(* IEC 61131-3 sources: eCockpitGit/test_project/src/%F%00 Library/%F%Common Functions/%F%Math/%F%Percent Difference, 2 files *)

(* ---- %POU%FU_diPerc_Diff.st ---- *)
//This function calculates the difference in percent between iA and iB, on the scale iMax
// +-----------+----------+----------+-----------------------------------------------------------------------------------------------------------------------+
// |**Version**|**Author**| **Date** |**Changes**                                                                                                            |
// +-----------+----------+----------+-----------------------------------------------------------------------------------------------------------------------+
// | 1         | NSN      | 11-12-18 | Creation                                                                                                              |
// +-----------+----------+----------+-----------------------------------------------------------------------------------------------------------------------+
FUNCTION FU_diPerc_Diff : DINT
VAR_INPUT
	iA		:DINT;
	iB		:DINT;
	iMax	:DINT;
END_VAR
(*%!%__DELIMITER__%!%*)
IF iA > iB THEN
	FU_diPerc_Diff	:=		(iA - iB) * 100 / iMax;
ELSE
	FU_diPerc_Diff	:=		(iB - iA) * 100 / iMax;
END_IF

(* ---- %POU%FU_iPerc_Diff.st ---- *)
//This function calculates the difference in percent between iA and iB, on the scale iMax
// +-----------+----------+----------+-----------------------------------------------------------------------------------------------------------------------+
// |**Version**|**Author**| **Date** |**Changes**                                                                                                            |
// +-----------+----------+----------+-----------------------------------------------------------------------------------------------------------------------+
// | 1         | NSN      | 10-01-18 | Updated to new format                                                                                                 |
// +-----------+----------+----------+-----------------------------------------------------------------------------------------------------------------------+
FUNCTION FU_iPerc_Diff : INT
VAR_INPUT
	iA		:INT;
	iB		:INT;
	iMax	:INT;
END_VAR
(*%!%__DELIMITER__%!%*)
IF iA > iB THEN
	FU_iPerc_Diff	:=		(iA - iB) * 100 / iMax;
ELSE
	FU_iPerc_Diff	:=		(iB - iA) * 100 / iMax;
END_IF
